{attribute 'pack_mode' := '2'}
TYPE U_XTS_TRANSPORT_STATE :
UNION
  stState             : ST_XTS_TRANSPORT_STATE;
  byState   AT %I*    : ARRAY[1..SIZEOF(ST_XTS_TRANSPORT_STATE)] OF BYTE;
END_UNION
END_TYPE

(* stored: Version 1.1.0.1
   DUT U_XTS_TRANSPORT_STATE: Id {26afc242-bfe9-4cd4-b584-d0100e5790c3} *)
